FUNCTION_BLOCK FB_Conveyor IMPLEMENTS I_Conveyor
VAR_OUTPUT
    bConveyorError        : BOOL;
    bConveyorMotorRun     : BOOL;
    bConveyorMotorReverse : BOOL;
END_VAR
VAR
    eMode       : E_ConveyorMode := E_ConveyorMode.IDLE;
    fbJamTimer  : TON;
END_VAR

//fbJamTimer(IN := bConveyorMotorRun, PT := GVL_Config.T_JAM_TIMEOUT);
IF fbJamTimer.Q THEN
    eMode := E_ConveyorMode.FAULT;
END_IF

CASE eMode OF
    E_ConveyorMode.IDLE:
        bConveyorMotorRun     := FALSE;
        bConveyorMotorReverse := FALSE;

    E_ConveyorMode.RUNNING_FORWARD:
        bConveyorMotorRun     := TRUE;
        bConveyorMotorReverse := FALSE;

    E_ConveyorMode.RUNNING_BACKWARD:
        bConveyorMotorRun     := TRUE;
        bConveyorMotorReverse := TRUE;

    E_ConveyorMode.FAULT:
        bConveyorMotorRun     := FALSE;
        bConveyorMotorReverse := FALSE;
        bConveyorError        := TRUE;
END_CASE

PROPERTY bError : BOOL
GET
bError := bConveyorError;
END_GET
END_PROPERTY

PROPERTY bMotorReverse : BOOL
GET
bMotorReverse := bConveyorMotorReverse;
END_GET
END_PROPERTY

PROPERTY bMotorRun : BOOL
GET
bMotorRun := bConveyorMotorRun;
END_GET
END_PROPERTY

METHOD M_Reset
VAR_INPUT
END_VAR
bConveyorError := FALSE;
eMode  := E_ConveyorMode.IDLE;
END_METHOD

METHOD M_Run
VAR_INPUT
    bForward : BOOL;
END_VAR
IF eMode = E_ConveyorMode.FAULT THEN
	RETURN;
END_IF
IF bForward THEN
    eMode := E_ConveyorMode.RUNNING_FORWARD;
ELSE
    eMode := E_ConveyorMode.RUNNING_BACKWARD;
END_IF
END_METHOD

METHOD M_Stop
VAR_INPUT
END_VAR
eMode := E_ConveyorMode.IDLE;
END_METHOD

END_FUNCTION_BLOCK

(* stored: Version 1.1.0.1, ProductVersion 3.1.4024.16
   POU FB_Conveyor: Id {ed03983f-d198-4ac9-879a-8e59f2a470c9}, SpecialFunc None
   Property bError: Id {aa000001-0000-0000-0000-000000000001}
   Get Get: Id {aa000002-0000-0000-0000-000000000001}
   Property bMotorReverse: Id {aa000005-0000-0000-0000-000000000001}
   Get Get: Id {aa000006-0000-0000-0000-000000000001}
   Property bMotorRun: Id {aa000003-0000-0000-0000-000000000001}
   Get Get: Id {aa000004-0000-0000-0000-000000000001}
   Method M_Reset: Id {aa000009-0000-0000-0000-000000000001}
   Method M_Run: Id {aa000007-0000-0000-0000-000000000001}
   Method M_Stop: Id {aa000008-0000-0000-0000-000000000001} *)
